TYPE ST_AnalogInput_Cfg :
STRUCT
    cfgScaleMin : REAL := 0.0;
    cfgScaleMax : REAL := 100.0;
END_STRUCT
END_TYPE

(* stored: Version 1.1.0.1, ProductVersion 3.1.4026.12
   DUT ST_AnalogInput_Cfg: Id {b0100003-0001-0000-0000-000000000001} *)
